(* Schneider Machine Expert - Basic project Contadores, file version 3.0.0.0 *)
(* ProjectInformations: Name=Contadores, Description=Exemplo de contadores para diversos tipos aplicados a automação industrial, usados para contagem de eventos até controle de processos. *)
(* UserInformations: LastName=Teodoro Araujo Junior, FirstName=Sidney, CellNumber=(27) 996489123, Email=sidneyteodoroaraujojunior2002@gmail.com, City=Belo Horizonte, State=Minas Gerais, Country=Brasil *)

HARDWARE
  Cpu 0: TM221M16R/G
  EthernetConfiguration: NetworkName=M221, IpAllocationMode=FixedAddress, IpAddress=0.0.0.0, SubnetMask=0.0.0.0
  SerialLineConfiguration: Baud=Baud19200, Parity=ParityEven, DataBits=DataBits8, StopBits=StopBits1, PhysicalMedium=PhysicalMediumRs485, TransmissionMode=TransmissionModeModbusRtu, SlaveId=1, Addressing=SlaveAddressing
  MastTask: UsePeriodScanMode=false, PeriodScan=100
  FastTask: Period=255
  CpuBehavior: StartingMode=StartAsPreviousState, AutoSaveRamOnEeprom=true, WatchdogPeriod=250

SYMBOLS  (address, symbol, comment, settings)
  %C0       CONTADOR_1  "Contador"  [Preset=5]
  %I0.0     RESET  "Resetar a contagem"
  %I0.1     PRESET  "Pre-definicao"
  %I0.2     ADICAO  "Incrementar contagem"
  %I0.3     SUBTRAI  "Decrementar contagem"
  %Q0.0     DECRESCENTE  "Sobrefluxo"
  %Q0.1     PRE_DEFINICAO  "Predefinicao atingida"
  %Q0.2     ASCENDENTE  "Contagem ascendente"

POU Novo POU
  (* SectionNumber=1 *)

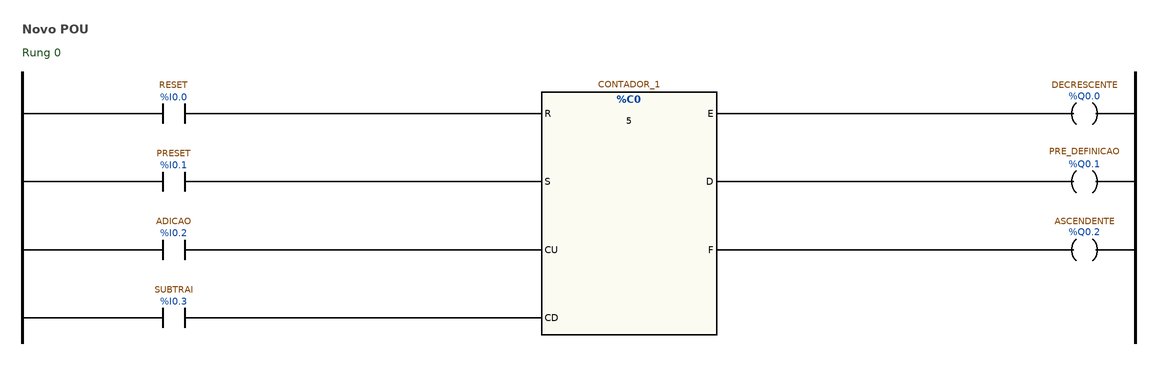

// Rung 0
  BLK %C0                 (* CONTADOR_1 *)
  LD %I0.0                (* RESET *)
  R
  LD %I0.1                (* PRESET *)
  S
  LD %I0.2                (* ADICAO *)
  CU
  LD %I0.3                (* SUBTRAI *)
  CD
  OUT_BLK
  LD E
  ST %Q0.0                (* DECRESCENTE *)
  LD D
  ST %Q0.1                (* PRE_DEFINICAO *)
  LD F
  ST %Q0.2                (* ASCENDENTE *)
  END_BLK
  // as ST:
  //   CONTADOR_1(R := RESET, S := PRESET, CU := ADICAO, CD := SUBTRAI);
  //   DECRESCENTE := CONTADOR_1.E;
  //   PRE_DEFINICAO := CONTADOR_1.D;
  //   ASCENDENTE := CONTADOR_1.F;
